{attribute 'GeneratedUsingTerminal: EL6001-0000-0020'}
{attribute addProperty BoxType "EL6001-0000-0020"}
{attribute addProperty Id "InputsAT %I*Inputs_E5D489814OutputsAT %Q*Outputs_1EA344054WcStateAT %I*WcState_9091E0EB2InfoDataAT %I*InfoData_32EB74EA10"}
{attribute addProperty CRC "2192288044"}
{attribute addProperty Size "20"}
TYPE EL6001_82ABA92C EXTENDS EtcSlaveTerminalBase_947E5A46 :
STRUCT
	{attribute addProperty Name "Inputs"}
	Inputs : Inputs_E5D48981;
	{attribute addProperty Name "Outputs"}
	Outputs : Outputs_1EA34405;
	{attribute addProperty Name "WcState"}
	WcState : WcState_9091E0EB;
	{attribute addProperty Name "InfoData"}
	InfoData : InfoData_32EB74EA;
END_STRUCT
END_TYPE

(* stored: Version 1.2.0.0, ProductVersion 3.1.4024.9
   DUT EL6001_82ABA92C: Id {2404df7a-a80e-40af-8d7e-54d5d6cbf7b4} *)
